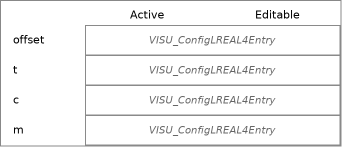
VISUALIZATION VISU_M2Config_ThermalFocusStation  // 342x147
VAR_IN_OUT
    editable : M2ThermalFocusStationConfig;
	active : M2ThermalFocusStationConfig;
END_VAR
    Label (85,5 125x20), "Active"
    Label (215,5 125x20), "Editable"
    Label (10,25 75x30), "offset"
    Label (10,55 70x30), "t"
    Label (10,85 75x30), "c"
    Label (10,115 75x30), "m"
    Frame (85,25 255x30)
        shows VISU_ConfigLREAL4Entry(active := active.offset, editable := editable.offset)
    Frame (85,55 255x30)
        shows VISU_ConfigLREAL4Entry(active := active.topCoefficient, editable := editable.topCoefficient)
    Frame (85,85 255x30)
        shows VISU_ConfigLREAL4Entry(active := active.centreCoefficient, editable := editable.centreCoefficient)
    Frame (85,115 255x30)
        shows VISU_ConfigLREAL4Entry(active := active.mirrorCellCoefficient, editable := editable.mirrorCellCoefficient)
END_VISUALIZATION

(* stored: Version 1.1.0.1, ProductVersion 3.1.4019.2
   Visu VISU_M2Config_ThermalFocusStation: Id {2ab8c076-83d7-4594-9f7d-3c7cbeac5d60} *)
